INTERFACE IEventHandler_OnDayChanged EXTENDS IEventHandlerBase

METHOD OnDayChanged
VAR_INPUT
	Now: TIMESTRUCT;
END_VAR
END_METHOD

END_INTERFACE

(* stored: Version 1.1.0.1, ProductVersion 3.1.4024.3
   Itf IEventHandler_OnDayChanged: Id {58c0c4e3-83ab-0c2a-26a0-804b3f758f7e}
   Method OnDayChanged: Id {d54ddf27-7a4f-0593-1289-301b5c20107b} *)
